// Gets the lower bound index of the array of specified type.
FUNCTION F_GetBoolArrayLowerBound : T_Position // The lower bound index of the specified array.
VAR_IN_OUT
	arArray : ARRAY[*] OF BOOL; // The array to query.
END_VAR

F_GetBoolArrayLowerBound := LOWER_BOUND(arArray, 1);

END_FUNCTION

(* stored: Version 1.1.0.1
   POU F_GetBoolArrayLowerBound: Id {2dd79da3-c3d0-0aa6-39a2-e1f0dbec617e}, SpecialFunc None *)
